(* LS Electric XG5000 project: 241011_연습_알람연동 *)
(* PLC LSPLC *)

PROGRAM NewProgram (* task: 스캔 프로그램 *)

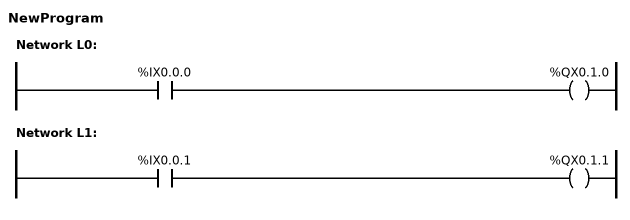
(* Rung L0 *)
%QX0.1.0 := %IX0.0.0;
(* Rung L1 *)
%QX0.1.1 := %IX0.0.1;
END_PROGRAM